// TIA Portal V17 export
// export: Created 2024-08-11T17:53:08.0637425Z, ExportSetting WithDefaults, DisplayName Totally Integrated Automation Portal, DisplayVersion V17 Update 5, DisplayName TIA Portal Openness, DisplayVersion V17 Update 5, DisplayName TIA Portal Version Control Interface, DisplayVersion V17, DisplayName SINAMICS Startdrive Advanced, DisplayVersion V17 SP1, DisplayName SINAMICS Startdrive G130, G150, S120, S150, SINAMICS MV, S210, DisplayVersion V17 SP1, DisplayName SINAMICS Startdrive G110M, G120, G120C, G120D, G120P, G115D, DisplayVersion V17 SP1, DisplayName STEP 7 Professional, DisplayVersion V17 Update 5, DisplayName STEP 7 Safety, DisplayVersion V17, DisplayName WinCC Advanced / Unified PC, DisplayVersion V17 Update 5
DATA_BLOCK "DB_ADDR"   // DB5
{ S7_Optimized_Access := 'FALSE' }
VERSION : 0.1
// stored: AutoNumber true, DBAccessibleFromOPCUA true, IsOnlyStoredInLoadMemory false, IsWriteProtectedInAS false
   VAR
      VOLT : UDInt := 48455;
      AMP : UDInt := 48453;
      FRE : UDInt := 48452;
      RPM : UDInt := 48456;
      SPEED : UDInt := 42331;
      RUN : UDInt := 42332;
      DIR : UDInt := 42333;
      OUT : UDInt;
   END_VAR
BEGIN
END_DATA_BLOCK
